// TIA Portal V17 export
// export: Created 2023-04-04T13:27:34.0477052Z, ExportSetting WithDefaults, DisplayName Totally Integrated Automation Portal, DisplayVersion V17, DisplayName TIA Portal Openness, DisplayVersion V17, DisplayName TIA Portal Version Control Interface, DisplayVersion V17, DisplayName STEP 7 Professional, DisplayVersion V17, DisplayName STEP 7 Safety, DisplayVersion V17, DisplayName WinCC Advanced, DisplayVersion V17
TYPE "typ_SPS_NFC_Module_State"
// stored: IsFailsafeCompliant false
   STRUCT
      ldt_ts : LDT;
      Workpiece : "typ_Workpiece";
      History { S7_SetPoint := 'True'} : Array[1..20] of "typ_History";
   END_STRUCT;
END_TYPE
